# EPICS substitutions: GALILMUL/GALILMUL-IOC-01App/Db/galil_digital_ports.substitutions
# Description:
# digital/binary port substitution file.
#
# This library is free software; you can redistribute it and/or
# modify it under the terms of the GNU Lesser General Public
# Licence as published by the Free Software Foundation; either
# version 2.1 of the Licence, or (at your option) any later version.
#
# This library is distributed in the hope that it will be useful,
# but WITHOUT ANY WARRANTY; without even the implied warranty of
# MERCHANTABILITY or FITNESS FOR A PARTICULAR PURPOSE.  See the GNU
# Lesser General Public Licence for more details.
#
# You should have received a copy of the GNU Lesser General Public
# Licence along with this library; if not, write to the Free Software
# Foundation, Inc., 51 Franklin St, Fifth Floor, Boston, MA 02110-1301 USA.
#
# Contact details:
# mark.clift@synchrotron.org.au
# 800 Blackburn Road, Clayton, Victoria 3168, Australia.
#

# P    - PV prefix
# R    - Record Name
# PORT - Asyn port name
# BYTE - Hardware byte to read
# MASK - Mask for this bit

file "$(GALIL)/GalilSup/Db/galil_digital_in_bit.template"
{
pattern {P,      R,          PORT,  BYTE,  MASK      }

# DMC = Digital motor controller
# DMC binary inputs are organized in bytes
	{\$(P):DMC\$(CCP),  Galil0Bi0,  "\$(PORT=Galil)", 0,     0x000001  }
	{\$(P):DMC\$(CCP),  Galil0Bi1,  "\$(PORT=Galil)", 0,     0x000002  }
	{\$(P):DMC\$(CCP),  Galil0Bi2,  "\$(PORT=Galil)", 0,     0x000004  }
	{\$(P):DMC\$(CCP),  Galil0Bi3,  "\$(PORT=Galil)", 0,     0x000008  }
	{\$(P):DMC\$(CCP),  Galil0Bi4,  "\$(PORT=Galil)", 0,     0x000010  }
	{\$(P):DMC\$(CCP),  Galil0Bi5,  "\$(PORT=Galil)", 0,     0x000020  }
	{\$(P):DMC\$(CCP),  Galil0Bi6,  "\$(PORT=Galil)", 0,     0x000040  }
	{\$(P):DMC\$(CCP),  Galil0Bi7,  "\$(PORT=Galil)", 0,     0x000080  }

	{\$(P):DMC\$(CCP),  Galil1Bi0,  "\$(PORT=Galil)", 1,     0x000001  }
	{\$(P):DMC\$(CCP),  Galil1Bi1,  "\$(PORT=Galil)", 1,     0x000002  }
	{\$(P):DMC\$(CCP),  Galil1Bi2,  "\$(PORT=Galil)", 1,     0x000004  }
	{\$(P):DMC\$(CCP),  Galil1Bi3,  "\$(PORT=Galil)", 1,     0x000008  }
	{\$(P):DMC\$(CCP),  Galil1Bi4,  "\$(PORT=Galil)", 1,     0x000010  }
	{\$(P):DMC\$(CCP),  Galil1Bi5,  "\$(PORT=Galil)", 1,     0x000020  }
	{\$(P):DMC\$(CCP),  Galil1Bi6,  "\$(PORT=Galil)", 1,     0x000040  }
	{\$(P):DMC\$(CCP),  Galil1Bi7,  "\$(PORT=Galil)", 1,     0x000080  }

}

# P    - PV prefix
# R    - Record Name
# PORT - Asyn port name
# WORD - Hardware word to read
# MASK - Mask for this bit

file "$(GALIL)/GalilSup/Db/galil_digital_out_bit.template"
{
pattern {P,      R,           PORT,  WORD,  MASK      }

# DMC binary outputs are organized in 16bit words
	{\$(P):DMC\$(CCP),  Galil0Bo0,   "\$(PORT=Galil)", 0,     0x000001  }
	{\$(P):DMC\$(CCP),  Galil0Bo1,   "\$(PORT=Galil)", 0,     0x000002  }
	{\$(P):DMC\$(CCP),  Galil0Bo2,   "\$(PORT=Galil)", 0,     0x000004  }
	{\$(P):DMC\$(CCP),  Galil0Bo3,   "\$(PORT=Galil)", 0,     0x000008  }
	{\$(P):DMC\$(CCP),  Galil0Bo4,   "\$(PORT=Galil)", 0,     0x000010  }
	{\$(P):DMC\$(CCP),  Galil0Bo5,   "\$(PORT=Galil)", 0,     0x000020  }
	{\$(P):DMC\$(CCP),  Galil0Bo6,   "\$(PORT=Galil)", 0,     0x000040  }
	{\$(P):DMC\$(CCP),  Galil0Bo7,   "\$(PORT=Galil)", 0,     0x000080  }
	{\$(P):DMC\$(CCP),  Galil0Bo8,   "\$(PORT=Galil)", 0,     0x000100  }
	{\$(P):DMC\$(CCP),  Galil0Bo9,   "\$(PORT=Galil)", 0,     0x000200  }
	{\$(P):DMC\$(CCP),  Galil0Bo10,  "\$(PORT=Galil)", 0,     0x000400  }
	{\$(P):DMC\$(CCP),  Galil0Bo11,  "\$(PORT=Galil)", 0,     0x000800  }
	{\$(P):DMC\$(CCP),  Galil0Bo12,  "\$(PORT=Galil)", 0,     0x001000  }
	{\$(P):DMC\$(CCP),  Galil0Bo13,  "\$(PORT=Galil)", 0,     0x002000  }
	{\$(P):DMC\$(CCP),  Galil0Bo14,  "\$(PORT=Galil)", 0,     0x004000  }
	{\$(P):DMC\$(CCP),  Galil0Bo15,  "\$(PORT=Galil)", 0,     0x008000  }

	{\$(P):DMC\$(CCP),  Galil1Bo0,   "\$(PORT=Galil)", 1,     0x000001  }
	{\$(P):DMC\$(CCP),  Galil1Bo1,   "\$(PORT=Galil)", 1,     0x000002  }
	{\$(P):DMC\$(CCP),  Galil1Bo2,   "\$(PORT=Galil)", 1,     0x000004  }
	{\$(P):DMC\$(CCP),  Galil1Bo3,   "\$(PORT=Galil)", 1,     0x000008  }
	{\$(P):DMC\$(CCP),  Galil1Bo4,   "\$(PORT=Galil)", 1,     0x000010  }
	{\$(P):DMC\$(CCP),  Galil1Bo5,   "\$(PORT=Galil)", 1,     0x000020  }
	{\$(P):DMC\$(CCP),  Galil1Bo6,   "\$(PORT=Galil)", 1,     0x000040  }
	{\$(P):DMC\$(CCP),  Galil1Bo7,   "\$(PORT=Galil)", 1,     0x000080  }
	{\$(P):DMC\$(CCP),  Galil1Bo8,   "\$(PORT=Galil)", 1,     0x000100  }
	{\$(P):DMC\$(CCP),  Galil1Bo9,   "\$(PORT=Galil)", 1,     0x000200  }
	{\$(P):DMC\$(CCP),  Galil1Bo10,  "\$(PORT=Galil)", 1,     0x000400  }
	{\$(P):DMC\$(CCP),  Galil1Bo11,  "\$(PORT=Galil)", 1,     0x000800  }
	{\$(P):DMC\$(CCP),  Galil1Bo12,  "\$(PORT=Galil)", 1,     0x001000  }
	{\$(P):DMC\$(CCP),  Galil1Bo13,  "\$(PORT=Galil)", 1,     0x002000  }
	{\$(P):DMC\$(CCP),  Galil1Bo14,  "\$(PORT=Galil)", 1,     0x004000  }
	{\$(P):DMC\$(CCP),  Galil1Bo15,  "\$(PORT=Galil)", 1,     0x008000  }

	{\$(P):DMC\$(CCP),  Galil2Bo0,   "\$(PORT=Galil)", 2,     0x000001  }
	{\$(P):DMC\$(CCP),  Galil2Bo1,   "\$(PORT=Galil)", 2,     0x000002  }
	{\$(P):DMC\$(CCP),  Galil2Bo2,   "\$(PORT=Galil)", 2,     0x000004  }
	{\$(P):DMC\$(CCP),  Galil2Bo3,   "\$(PORT=Galil)", 2,     0x000008  }
	{\$(P):DMC\$(CCP),  Galil2Bo4,   "\$(PORT=Galil)", 2,     0x000010  }
	{\$(P):DMC\$(CCP),  Galil2Bo5,   "\$(PORT=Galil)", 2,     0x000020  }
	{\$(P):DMC\$(CCP),  Galil2Bo6,   "\$(PORT=Galil)", 2,     0x000040  }
	{\$(P):DMC\$(CCP),  Galil2Bo7,   "\$(PORT=Galil)", 2,     0x000080  }
	{\$(P):DMC\$(CCP),  Galil2Bo8,   "\$(PORT=Galil)", 2,     0x000100  }
	{\$(P):DMC\$(CCP),  Galil2Bo9,   "\$(PORT=Galil)", 2,     0x000200  }
	{\$(P):DMC\$(CCP),  Galil2Bo10,  "\$(PORT=Galil)", 2,     0x000400  }
	{\$(P):DMC\$(CCP),  Galil2Bo11,  "\$(PORT=Galil)", 2,     0x000800  }
	{\$(P):DMC\$(CCP),  Galil2Bo12,  "\$(PORT=Galil)", 2,     0x001000  }
	{\$(P):DMC\$(CCP),  Galil2Bo13,  "\$(PORT=Galil)", 2,     0x002000  }
	{\$(P):DMC\$(CCP),  Galil2Bo14,  "\$(PORT=Galil)", 2,     0x004000  }
	{\$(P):DMC\$(CCP),  Galil2Bo15,  "\$(PORT=Galil)", 2,     0x008000  }

	{\$(P):DMC\$(CCP),  Galil3Bo0,   "\$(PORT=Galil)", 3,     0x000001  }
	{\$(P):DMC\$(CCP),  Galil3Bo1,   "\$(PORT=Galil)", 3,     0x000002  }
	{\$(P):DMC\$(CCP),  Galil3Bo2,   "\$(PORT=Galil)", 3,     0x000004  }
	{\$(P):DMC\$(CCP),  Galil3Bo3,   "\$(PORT=Galil)", 3,     0x000008  }
	{\$(P):DMC\$(CCP),  Galil3Bo4,   "\$(PORT=Galil)", 3,     0x000010  }
	{\$(P):DMC\$(CCP),  Galil3Bo5,   "\$(PORT=Galil)", 3,     0x000020  }
	{\$(P):DMC\$(CCP),  Galil3Bo6,   "\$(PORT=Galil)", 3,     0x000040  }
	{\$(P):DMC\$(CCP),  Galil3Bo7,   "\$(PORT=Galil)", 3,     0x000080  }
	{\$(P):DMC\$(CCP),  Galil3Bo8,   "\$(PORT=Galil)", 3,     0x000100  }
	{\$(P):DMC\$(CCP),  Galil3Bo9,   "\$(PORT=Galil)", 3,     0x000200  }
	{\$(P):DMC\$(CCP),  Galil3Bo10,  "\$(PORT=Galil)", 3,     0x000400  }
	{\$(P):DMC\$(CCP),  Galil3Bo11,  "\$(PORT=Galil)", 3,     0x000800  }
	{\$(P):DMC\$(CCP),  Galil3Bo12,  "\$(PORT=Galil)", 3,     0x001000  }
	{\$(P):DMC\$(CCP),  Galil3Bo13,  "\$(PORT=Galil)", 3,     0x002000  }
	{\$(P):DMC\$(CCP),  Galil3Bo14,  "\$(PORT=Galil)", 3,     0x004000  }
	{\$(P):DMC\$(CCP),  Galil3Bo15,  "\$(PORT=Galil)", 3,     0x008000  }

	{\$(P):DMC\$(CCP),  Galil4Bo0,   "\$(PORT=Galil)", 4,     0x000001  }
	{\$(P):DMC\$(CCP),  Galil4Bo1,   "\$(PORT=Galil)", 4,     0x000002  }
	{\$(P):DMC\$(CCP),  Galil4Bo2,   "\$(PORT=Galil)", 4,     0x000004  }
	{\$(P):DMC\$(CCP),  Galil4Bo3,   "\$(PORT=Galil)", 4,     0x000008  }
	{\$(P):DMC\$(CCP),  Galil4Bo4,   "\$(PORT=Galil)", 4,     0x000010  }
	{\$(P):DMC\$(CCP),  Galil4Bo5,   "\$(PORT=Galil)", 4,     0x000020  }
	{\$(P):DMC\$(CCP),  Galil4Bo6,   "\$(PORT=Galil)", 4,     0x000040  }
	{\$(P):DMC\$(CCP),  Galil4Bo7,   "\$(PORT=Galil)", 4,     0x000080  }
	{\$(P):DMC\$(CCP),  Galil4Bo8,   "\$(PORT=Galil)", 4,     0x000100  }
	{\$(P):DMC\$(CCP),  Galil4Bo9,   "\$(PORT=Galil)", 4,     0x000200  }
	{\$(P):DMC\$(CCP),  Galil4Bo10,  "\$(PORT=Galil)", 4,     0x000400  }
	{\$(P):DMC\$(CCP),  Galil4Bo11,  "\$(PORT=Galil)", 4,     0x000800  }
	{\$(P):DMC\$(CCP),  Galil4Bo12,  "\$(PORT=Galil)", 4,     0x001000  }
	{\$(P):DMC\$(CCP),  Galil4Bo13,  "\$(PORT=Galil)", 4,     0x002000  }
	{\$(P):DMC\$(CCP),  Galil4Bo14,  "\$(PORT=Galil)", 4,     0x004000  }
	{\$(P):DMC\$(CCP),  Galil4Bo15,  "\$(PORT=Galil)", 4,     0x008000  }

}

# end
